// TIA Portal V17 export
// export: Created 2023-04-11T09:34:01.7220227Z, ExportSetting WithDefaults, DisplayName Totally Integrated Automation Portal, DisplayVersion V17 Update 3, DisplayName TIA Portal Openness, DisplayVersion V17 Update 3, DisplayName TIA Portal Version Control Interface, DisplayVersion V17, DisplayName SINAMICS Startdrive Advanced, DisplayVersion V17 Update2, DisplayName SINAMICS Startdrive G130, G150, S120, S150, SINAMICS MV, S210, DisplayVersion V17 Update2, DisplayName SINAMICS Startdrive G110M, G120, G120C, G120D, G120P, G115D, DisplayVersion V17 Update2, DisplayName STEP 7 Professional, DisplayVersion V17 Update 3, DisplayName STEP 7 Safety, DisplayVersion V17, DisplayName WinCC UA Professional, DisplayVersion V17 Update 3
FUNCTION "FC_controlReadData_1" : Void   // FC19, LAD
{ S7_Optimized_Access := 'TRUE' }
VERSION : 0.1
// stored: AutoNumber true, IsIECCheckEnabled false, SetENOAutomatically false, UDAEnableTagReadback false
   VAR_INPUT
      header : String;
      footer : String;
   END_VAR
   VAR_IN_OUT
      IN : "t_LString";
      OUT : "t_LString";
   END_VAR
   VAR_TEMP
      headerPos : UInt;
      footerPos : UInt;
      ftrLen : UInt;
   END_VAR
BEGIN

REGION Network 1 (SCL)
   ENO := false;
   #ftrLen := INT_TO_UINT(LEN(#footer));

   #headerPos:="FIND_LS_S_1"(IN1:=#IN, IN2:=#header);

   IF #headerPos > 0 THEN
       "SUBSTR_LS_LS_2"(IN := #IN,
                      P := #headerPos + 1,
                      L := "LEN_LS_1"(#IN)-(#headerPos),
                      OUT := #OUT);
   ELSE
       RETURN;
   END_IF;


   #footerPos := "FIND_LS_S_1"(IN1 := #OUT, IN2 := #footer);

   IF #footerPos > 0 THEN
       #OUT.Len := #footerPos - #ftrLen;
       ENO := true;
   ELSE
       "CLEAR_LS_1"(#OUT);
   END_IF;
END_REGION
END_FUNCTION
